// TIA Portal V19 export
DATA_BLOCK "PIDHmiInterfaceDB"   // DB9
{ S7_Optimized_Access := 'TRUE' }
// stored: AutoNumber false, MemoryReserve 0
   VAR RETAIN
      M0940 : "M0940_HmiInterface";
   END_VAR
BEGIN
   M0940.PV := 0.0;
   M0940.SP := 0.0;
   M0940.EngUnitsMin := 0.0;
   M0940.EngUnitsMax := 0.0;
   M0940.P := 0.0;
   M0940.MV := 0.0;
   M0940.OP := 0.0;
END_DATA_BLOCK
